TYPE
    linked_racks_typ : STRUCT
        first_linked_rack  : INT;
        second_linked_rack : INT;
    END_STRUCT
END_TYPE

(* stored: Version 1.1.0.1
   DUT linked_racks_typ: Id {94c83ed1-82f8-4bfd-846b-23a2aee63f31} *)
